FUNCTION F_SAFETY_StatusFB_TO_MON : ST_SAFETY_FBMON
VAR_INPUT
	stFBStatus						: ST_SAFETY_FBStatus; 	(* Struktura ogolna *)
END_VAR

F_SAFETY_StatusFB_TO_MON.uStatus.stStatusWords	:= stFBStatus;									(* Przepisanie *)
F_SAFETY_StatusFB_TO_MON.eState 				:= stFBStatus.BState;							(* Ustawienie enum *)
F_SAFETY_StatusFB_TO_MON.bGeneralError			:= stFBStatus.wDiagnosis <> 0;					(* General Error *)

END_FUNCTION

(* stored: Version 1.1.0.1, ProductVersion 3.1.4022.12
   POU F_SAFETY_StatusFB_TO_MON: Id {73c35747-3c66-4a30-8c3e-a37ebf14c627}, SpecialFunc None *)
